FUNCTION_BLOCK ABSTRACT RFC_MoveWorkpiece_Base EXTENDS ControlPrimitiveBase
VAR_INPUT
END_VAR
VAR_OUTPUT
END_VAR
VAR
	m_ptrRFC: POINTER TO RefeedingConveyor;
	
	m_step: INT := 0;
END_VAR

SUPER^();

METHOD  Abort : BOOL
VAR_INPUT
END_VAR
m_ptrRFC^.METH_ConveyorStop();
m_ptrRFC^.METH_Switch_Retract();
Abort := TRUE;
END_METHOD

METHOD PROTECTED ABSTRACT AtTarget : BOOL
VAR_INPUT
END_VAR
END_METHOD

(* Execution logic of this Control Primitive. *)
METHOD PROTECTED ExecuteInternal : BOOL
VAR_INPUT
	i_params: ParameterSet;
END_VAR
CASE m_step OF
	0: // to target	
	IF NOT AtTarget() THEN
		m_ptrRFC^.METH_ConveyorForward();
		m_step := 1;
	END_IF
		
	1:
	IF AtTarget() THEN
		m_ptrRFC^.METH_ConveyorStop();
		//m_ptrPAC^.METH_Switch_Extend();
		m_step := 0;
		ExecuteInternal := TRUE;
	END_IF
		
END_CASE
END_METHOD

END_FUNCTION_BLOCK

(* stored: Version 1.1.0.1
   POU RFC_MoveWorkpiece_Base: Id {e5d5e346-e1b8-41a8-b595-fbdd0a35e3db}, SpecialFunc None
   Method Abort: Id {2f29c146-5e26-43a3-9487-b10b9cbea838}
   Method AtTarget: Id {f0bbd90a-dbe3-4759-9f7d-359f5d9b7d48}
   Method ExecuteInternal: Id {e3519d3b-4387-4208-9252-a3240bee6252} *)
